{attribute 'qualified_only'}
{attribute 'strict'}
TYPE E_Modes :
(
	Off,
	Auto,
	Manual
);
END_TYPE

(* stored: Version 1.1.0.1, ProductVersion 3.1.4024.12
   DUT Modes: Id {8bc1499c-d72b-4047-be06-7046324cc44f} *)
